Omron CX-Programmer project NewProject (CX-Programmer 9.73)

# PLC NewPLC1: CP1L M

## Global symbols (name address type ; comment)
100.04 BOOL  ; YELLOW_LIGHT_WAY_2
100.03 BOOL  ; RED_LIGHT_WAY_2
T0001 BOOL  ; T1
0.00 BOOL  ; ON_START
0.01 BOOL  ; OFF_BUTTON
0.03 BOOL  ; EMERGENCY_BUTTON
100.00 BOOL  ; RED_LIGHT_WAY_1
100.01 BOOL  ; YELLOW_LIGHT_WAY_1
100.02 BOOL  ; GREEN_LIGHT_WAY_1
100.05 BOOL  ; GREEN_LIGHT_WAY_2
100.06 BOOL  ; RED_LIGHT_WAY_3
100.07 BOOL  ; YELLOW_LIGHT_WAY_3
100.08 BOOL  ; GREEN_LIGHT_WAY_3
100.09 BOOL  ; RED_LIGHT_WAY_4
100.10 BOOL  ; YELLOW_LIGHT_WAY_4
100.11 BOOL  ; GREEN_LIGHT_WAY_4
C0001 BOOL  ; C1
C0002 BOOL  ; C2
C0003 BOOL  ; C3
C0004 BOOL  ; C4
T0000 BOOL  ; DELAY OFF
T0002 BOOL  ; T2
T0003 BOOL  ; T3
T0004 BOOL  ; T4
T0010 BOOL  ; STARTER _DELAY
W100.00 BOOL  ; 0
W100.03 BOOL  ; EMERGENCY

## Program NewProgram1 (cyclic task 0)

### Section Section1

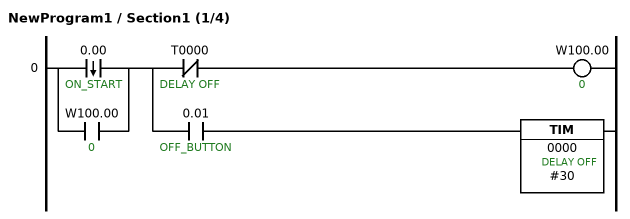
; rung 0
%LD 0.00  ; ON_START
OR W100.00  ; 0
OUT TR0
ANDNOT T0000  ; DELAY OFF
OUT W100.00  ; 0
LD TR0
AND 0.01  ; OFF_BUTTON
TIM 0000 #30  ; DELAY OFF

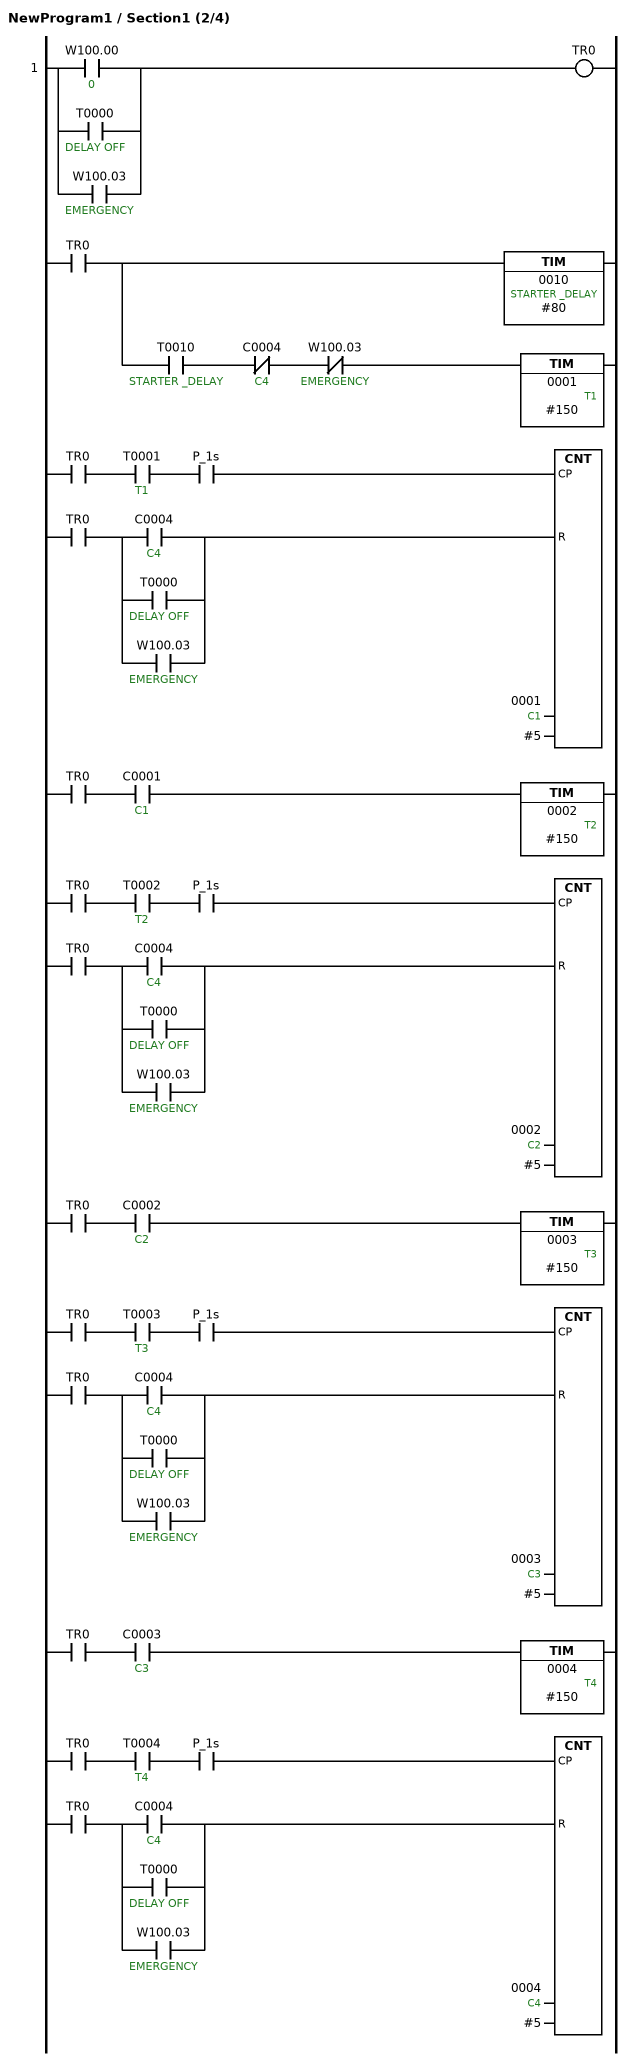
; rung 1
LD W100.00  ; 0
OR T0000  ; DELAY OFF
OR W100.03  ; EMERGENCY
OUT TR0
TIM 0010 #80  ; STARTER _DELAY
AND T0010  ; STARTER _DELAY
ANDNOT C0004  ; C4
ANDNOT W100.03  ; EMERGENCY
TIM 0001 #150  ; T1
LD TR0
AND T0001  ; T1
AND P_1s
LD TR0
LD C0004  ; C4
OR T0000  ; DELAY OFF
OR W100.03  ; EMERGENCY
ANDLD
CNT 0001 #5  ; C1
LD TR0
AND C0001  ; C1
TIM 0002 #150  ; T2
LD TR0
AND T0002  ; T2
AND P_1s
LD TR0
LD C0004  ; C4
OR T0000  ; DELAY OFF
OR W100.03  ; EMERGENCY
ANDLD
CNT 0002 #5  ; C2
LD TR0
AND C0002  ; C2
TIM 0003 #150  ; T3
LD TR0
AND T0003  ; T3
AND P_1s
LD TR0
LD C0004  ; C4
OR T0000  ; DELAY OFF
OR W100.03  ; EMERGENCY
ANDLD
CNT 0003 #5  ; C3
LD TR0
AND C0003  ; C3
TIM 0004 #150  ; T4
LD TR0
AND T0004  ; T4
AND P_1s
LD TR0
LD C0004  ; C4
OR T0000  ; DELAY OFF
OR W100.03  ; EMERGENCY
ANDLD
CNT 0004 #5  ; C4

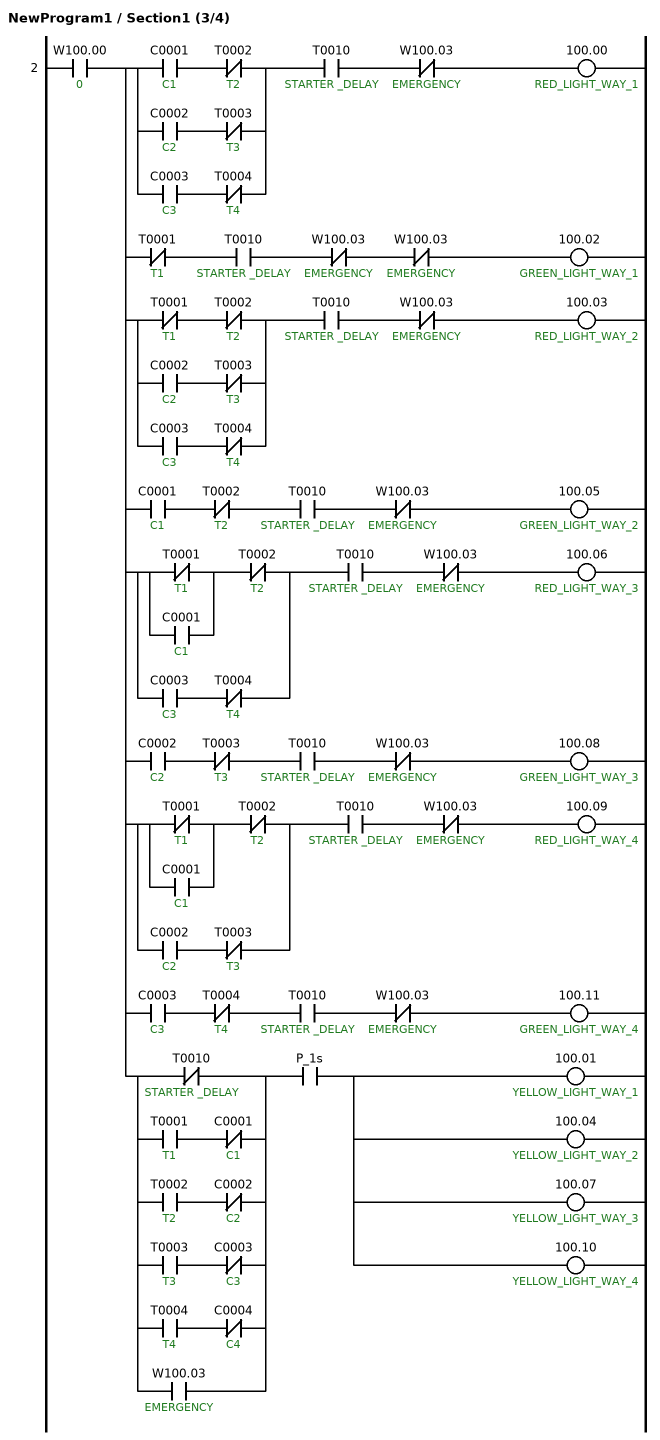
; rung 2
LD W100.00  ; 0
OUT TR0
LD C0001  ; C1
ANDNOT T0002  ; T2
LD C0002  ; C2
ANDNOT T0003  ; T3
ORLD
LD C0003  ; C3
ANDNOT T0004  ; T4
ORLD
ANDLD
AND T0010  ; STARTER _DELAY
ANDNOT W100.03  ; EMERGENCY
OUT 100.00  ; RED_LIGHT_WAY_1
LD TR0
ANDNOT T0001  ; T1
AND T0010  ; STARTER _DELAY
ANDNOT W100.03  ; EMERGENCY
ANDNOT W100.03  ; EMERGENCY
OUT 100.02  ; GREEN_LIGHT_WAY_1
LD TR0
LDNOT T0001  ; T1
ANDNOT T0002  ; T2
LD C0002  ; C2
ANDNOT T0003  ; T3
ORLD
LD C0003  ; C3
ANDNOT T0004  ; T4
ORLD
ANDLD
AND T0010  ; STARTER _DELAY
ANDNOT W100.03  ; EMERGENCY
OUT 100.03  ; RED_LIGHT_WAY_2
LD TR0
AND C0001  ; C1
ANDNOT T0002  ; T2
AND T0010  ; STARTER _DELAY
ANDNOT W100.03  ; EMERGENCY
OUT 100.05  ; GREEN_LIGHT_WAY_2
LD TR0
LDNOT T0001  ; T1
OR C0001  ; C1
ANDNOT T0002  ; T2
LD C0003  ; C3
ANDNOT T0004  ; T4
ORLD
ANDLD
AND T0010  ; STARTER _DELAY
ANDNOT W100.03  ; EMERGENCY
OUT 100.06  ; RED_LIGHT_WAY_3
LD TR0
AND C0002  ; C2
ANDNOT T0003  ; T3
AND T0010  ; STARTER _DELAY
ANDNOT W100.03  ; EMERGENCY
OUT 100.08  ; GREEN_LIGHT_WAY_3
LD TR0
LDNOT T0001  ; T1
OR C0001  ; C1
ANDNOT T0002  ; T2
LD C0002  ; C2
ANDNOT T0003  ; T3
ORLD
ANDLD
AND T0010  ; STARTER _DELAY
ANDNOT W100.03  ; EMERGENCY
OUT 100.09  ; RED_LIGHT_WAY_4
LD TR0
AND C0003  ; C3
ANDNOT T0004  ; T4
AND T0010  ; STARTER _DELAY
ANDNOT W100.03  ; EMERGENCY
OUT 100.11  ; GREEN_LIGHT_WAY_4
LD TR0
LDNOT T0010  ; STARTER _DELAY
LD T0001  ; T1
ANDNOT C0001  ; C1
ORLD
LD T0002  ; T2
ANDNOT C0002  ; C2
ORLD
LD T0003  ; T3
ANDNOT C0003  ; C3
ORLD
LD T0004  ; T4
ANDNOT C0004  ; C4
ORLD
OR W100.03  ; EMERGENCY
ANDLD
AND P_1s
OUT 100.01  ; YELLOW_LIGHT_WAY_1
OUT 100.04  ; YELLOW_LIGHT_WAY_2
OUT 100.07  ; YELLOW_LIGHT_WAY_3
OUT 100.10  ; YELLOW_LIGHT_WAY_4

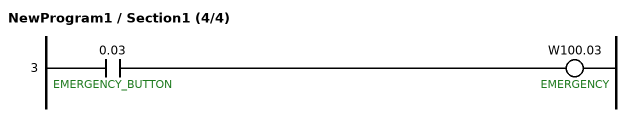
; rung 3
LD 0.03  ; EMERGENCY_BUTTON
OUT W100.03  ; EMERGENCY

### Section END
; rung 0
END(001)